Fanuc KAREL source: kt00069.KL

-- PROVISIONAL review KL for V1013-1; original PC SHA256 968aeb2bc5ed7e9988eab51b71758ffaafeba0ffde15e0ee24d6f3ea72f7fb14
-- Incomplete behavior may be omitted. Consult companion uncertainty JSON. Do not deploy.
PROGRAM KT00069
%NOLOCKGROUP
VAR
  I1 : INTEGER
  OUT : INTEGER
-- UNRESOLVED_DECL Y2 type=002018
BEGIN
  -- UNRESOLVED_PC offsets 5-16; opcodes 2E,23
  -- UNRESOLVED_PC offsets 21-35; opcodes 2E,22,9D,33,B2
  -- UNRESOLVED_PC offsets 40-62; opcodes 21,22,9D,33,B1,54,23
  -- UNRESOLVED_PC offsets 67-71; opcodes 7F
END KT00069
